// TIA Portal V20 export
DATA_BLOCK "FSIDB_Main_Safety_RTG1"   // DB1, F_DB
NAME : FUSI
// stored: InstanceOfName FSFB_Main_Safety_RTG1, InstanceOfType FB
"FSFB_Main_Safety_RTG1"
   // VAR
   //    AllStopZone1 { ExternalAccessible := 'False'; ExternalVisible := 'False'; ExternalWritable := 'False'} : Bool;
   //    AllStopZone2 : Bool;
   //    Reset : Bool;
   //    Pair1 : ESTOP1;
   //    Pair2 : ESTOP1;
   //    Pair3 : ESTOP1;
   //    Pair4 : ESTOP1;
   //    Pair5 : ESTOP1;
   //    Pair6 : ESTOP1;
   //    Pair7 : ESTOP1;
   //    Pair8 : ESTOP1;
   //    Pair9 : ESTOP1;
   //    Pair10 : ESTOP1;
   //    ACK_GL : ACK_GL;
   //    ResetDelayTimer_Pair1 : TOF;
   //    ResetDelayTimer_Pair2 : TOF;
   //    ResetDelayTimer_Pair3 : TOF;
   //    ResetDelayTimer_Pair4 : TOF;
   //    ResetDelayTimer_Pair5 : TOF;
   //    ResetDelayTimer_Pair6 : TOF;
   //    ResetDelayTimer_Pair7 : TOF;
   //    ResetDelayTimer_Pair8 : TOF;
   //    ResetDelayTimer_Pair9 : TOF;
   //    ResetDelayTimer_Pair10 : TOF;
   //    mem_Pair1 : Bool;
   //    mem_Pair2 : Bool;
   //    mem_Pair3 : Bool;
   //    mem_Pair4 : Bool;
   //    mem_Pair5 : Bool;
   //    mem_Pair6 : Bool;
   //    mem_Pair7 : Bool;
   //    mem_Pair8 : Bool;
   //    mem_Pair9 : Bool;
   //    mem_Pair10 : Bool;
   // END_VAR
BEGIN
END_DATA_BLOCK
